TYPE
    IdentityCoe :
    STRUCT
        VendorId : DWORD;
        ProductKey   : DWORD;
        Revision     : DWORD;
        SerialNumber : DWORD;
    END_STRUCT
END_TYPE

(* stored: Version 1.1.0.1, ProductVersion 3.1.4024.12
   DUT IdentityCoe: Id {584af156-93fd-44fd-acc0-2ddff86e5554} *)
